(* IEC 61131-3 sources: repolevel_ST_code_completion/real_groud_truth最新/repoeval_plc_hello_mixing_tank/full_result, 6 files *)

(* ---- F_ResetDeviceCommands.st ---- *)
FUNCTION F_ResetDeviceCommands : BOOL
VAR_IN_OUT
	// HMI命令标志（需要复位）
	bMixerRunCmd		:	BOOL;
	bMixerStopCmd		:	BOOL;
	bMedium1OpenCmd		:	BOOL;
	bMedium1CloseCmd	:	BOOL;
	bMedium2OpenCmd		:	BOOL;
	bMedium2CloseCmd	:	BOOL;
	bDrainOpenCmd		:	BOOL;
	bDrainCloseCmd		:	BOOL;
END_VAR
VAR_INPUT
	// 设备状态反馈
	bMixerRunning		:	BOOL;
	bMedium1Opened		:	BOOL;
	bMedium2Opened		:	BOOL;
	bDrainOpened		:	BOOL;
END_VAR

VAR_OUTPUT
	// 复位完成标志
	bResetComplete		:	BOOL;
END_VAR

// 功能描述：复位所有HMI命令标志，当设备状态与命令一致时完成复位
bResetComplete := FALSE;

// 混合电机命令复位逻辑
IF NOT bMixerRunning AND bMixerRunCmd THEN
	bMixerRunCmd := FALSE;
END_IF;

IF bMixerRunning AND bMixerStopCmd THEN
	bMixerStopCmd := FALSE;
END_IF;

// Medium1命令复位逻辑
IF NOT bMedium1Opened AND bMedium1OpenCmd THEN
	bMedium1OpenCmd := FALSE;
END_IF;

IF bMedium1Opened AND bMedium1CloseCmd THEN
	bMedium1CloseCmd := FALSE;
END_IF;

// Medium2命令复位逻辑
IF NOT bMedium2Opened AND bMedium2OpenCmd THEN
	bMedium2OpenCmd := FALSE;
END_IF;

IF bMedium2Opened AND bMedium2CloseCmd THEN
	bMedium2CloseCmd := FALSE;
END_IF;

// Drain命令复位逻辑
IF NOT bDrainOpened AND bDrainOpenCmd THEN
	bDrainOpenCmd := FALSE;
END_IF;

IF bDrainOpened AND bDrainCloseCmd THEN
	bDrainCloseCmd := FALSE;
END_IF;

// 检查是否所有命令标志已复位
IF NOT bMixerRunCmd AND NOT bMixerStopCmd AND
   NOT bMedium1OpenCmd AND NOT bMedium1CloseCmd AND
   NOT bMedium2OpenCmd AND NOT bMedium2CloseCmd AND
   NOT bDrainOpenCmd AND NOT bDrainCloseCmd THEN
	bResetComplete := TRUE;
END_IF;

RETURN bResetComplete;
END_FUNCTION

(* ---- F_UpdateLimitSwitches.st ---- *)
FUNCTION F_UpdateLimitSwitches : BOOL
VAR_INPUT
	rTankLevel			:	REAL;			// 当前液位 (%)
	rFullThreshold		:	REAL := 85.0;	// 满液位阈值 (%)
	rEmptyThreshold		:	REAL := 5.0;	// 空液位阈值 (%)
END_VAR
VAR_OUTPUT
	bLevelFull			:	BOOL;			// 液位满开关
	bLevelEmpty			:	BOOL;			// 液位空开关
END_VAR

# --------------------------------------------------
# FUNCTION F_UpdateLimitSwitches
# This function updates the limit switches based on the current tank level.
# If the tank level exceeds the full threshold, the full switch is activated.
# If the tank level drops below the empty threshold, the empty switch is activated.
# --------------------------------------------------

# Update the full level switch
IF rTankLevel >= rFullThreshold THEN
    bLevelFull := TRUE;
ELSE
    bLevelFull := FALSE;
END_IF;

# Update the empty level switch
IF rTankLevel <= rEmptyThreshold THEN
    bLevelEmpty := TRUE;
ELSE
    bLevelEmpty := FALSE;
END_IF;

# Return TRUE to indicate the function executed successfully
F_UpdateLimitSwitches := TRUE;
END_FUNCTION

(* ---- FB_AutoSequence.st ---- *)
FUNCTION_BLOCK FB_AutoSequence
VAR_INPUT
	bEnable				:	BOOL;			// 使能自动序列
	bReset				:	BOOL;			// 复位到排空状态

	// 液位传感器反馈
	bTankLevelFull		:	BOOL;			// 液位满传感器
	bTankLevelEmpty		:	BOOL;			// 液位空传感器

	// 设备状态反馈
	bMixerRunning		:	BOOL;			// 混合电机运行中
	bMedium1Opened		:	BOOL;			// 介质1阀门打开
	bMedium2Opened		:	BOOL;			// 介质2阀门打开
	bDrainOpened		:	BOOL;			// 排空阀门打开

	// 配置参数
	tMixingDuration		:	TIME := T#10S;	// 混合持续时间
END_VAR
VAR_OUTPUT
	// 设备控制输出
	bMixerRunCmd		:	BOOL;			// 混合电机运行命令
	bMedium1OpenCmd		:	BOOL;			// 介质1阀门打开命令
	bMedium2OpenCmd		:	BOOL;			// 介质2阀门打开命令
	bDrainOpenCmd		:	BOOL;			// 排空阀门打开命令

	// 状态输出
	eCurrentState		:	AUTO_SEQUENCE;	// 当前状态
	nCyclesCompleted	:	UINT;			// 完成的循环次数
END_VAR

VAR
	// 内部状态变量
	eNextState			:	AUTO_SEQUENCE;	// 下一个状态
	tStateTimer			:	TIME;			// 状态计时器
	nCycleCounter		:	UINT := 0;		// 循环计数器
	bTransitionFlag		:	BOOL := FALSE;	// 状态转换标志
END_VAR

// 自动序列状态枚举
TYPE AUTO_SEQUENCE :
(
	IDLE,				// 空闲状态
	FILLING_MEDIUM1,	// 介质1填充状态
	FILLING_MEDIUM2,	// 介质2填充状态
	MIXING,				// 混合状态
	DRAINING			// 排空状态
);
END_TYPE

// 自动序列逻辑实现
IF bEnable THEN
	CASE eCurrentState OF
		IDLE:
			IF bTankLevelEmpty THEN
				eNextState := FILLING_MEDIUM1;
			END_IF;

		FILLING_MEDIUM1:
			bMedium1OpenCmd := TRUE;
			IF bTankLevelFull THEN
				bMedium1OpenCmd := FALSE;
				eNextState := FILLING_MEDIUM2;
			END_IF;

		FILLING_MEDIUM2:
			bMedium2OpenCmd := TRUE;
			IF bTankLevelFull THEN
				bMedium2OpenCmd := FALSE;
				eNextState := MIXING;
			END_IF;

		MIXING:
			bMixerRunCmd := TRUE;
			IF tStateTimer >= tMixingDuration THEN
				bMixerRunCmd := FALSE;
				eNextState := DRAINING;
			END_IF;

		DRAINING:
			bDrainOpenCmd := TRUE;
			IF bTankLevelEmpty THEN
				bDrainOpenCmd := FALSE;
				eNextState := IDLE;
				nCycleCounter := nCycleCounter + 1;
			END_IF;
	END_CASE;

	// 状态更新
	IF eNextState <> eCurrentState THEN
		eCurrentState := eNextState;
		tStateTimer := T#0S; // 重置状态计时器
	END_IF;

	// 状态计时器更新
	tStateTimer := tStateTimer + T#1MS;
ELSE
	// 禁用时复位所有命令和状态
	bMixerRunCmd := FALSE;
	bMedium1OpenCmd := FALSE;
	bMedium2OpenCmd := FALSE;
	bDrainOpenCmd := FALSE;
	eCurrentState := IDLE;
	nCycleCounter := 0;
END_IF;

IF bReset THEN
	// 复位逻辑
	bMixerRunCmd := FALSE;
	bMedium1OpenCmd := FALSE;
	bMedium2OpenCmd := FALSE;
	bDrainOpenCmd := FALSE;
	eCurrentState := IDLE;
	nCycleCounter := 0;
	tStateTimer := T#0S;
END_IF;
END_FUNCTION_BLOCK

(* ---- FB_ManualControl.st ---- *)
FUNCTION_BLOCK FB_ManualControl
VAR_INPUT
	// HMI命令输入
	bMixerRunCmd		:	BOOL;
	bMixerStopCmd		:	BOOL;
	bMedium1OpenCmd		:	BOOL;
	bMedium1CloseCmd	:	BOOL;
	bMedium2OpenCmd		:	BOOL;
	bMedium2CloseCmd	:	BOOL;
	bDrainOpenCmd		:	BOOL;
	bDrainCloseCmd		:	BOOL;

	// 设备反馈输入
	bMixerRunning		:	BOOL;
	bMedium1Opened		:	BOOL;
	bMedium2Opened		:	BOOL;
	bDrainOpened		:	BOOL;
END_VAR
VAR_OUTPUT
	// 设备控制输出
	bMixerRunCmdOut		:	BOOL;
	bMedium1OpenCmdOut	:	BOOL;
	bMedium2OpenCmdOut	:	BOOL;
	bDrainOpenCmdOut	:	BOOL;
END_VAR

VAR
	// 内部变量
	bResetCommands		:	BOOL;
END_VAR

// 主程序逻辑
// 复位命令逻辑
bResetCommands := F_ResetDeviceCommands(
	bMixerRunCmd := bMixerRunCmd,
	bMixerStopCmd := bMixerStopCmd,
	bMedium1OpenCmd := bMedium1OpenCmd,
	bMedium1CloseCmd := bMedium1CloseCmd,
	bMedium2OpenCmd := bMedium2OpenCmd,
	bMedium2CloseCmd := bMedium2CloseCmd,
	bDrainOpenCmd := bDrainOpenCmd,
	bDrainCloseCmd := bDrainCloseCmd,
	bMixerRunning := bMixerRunning,
	bMedium1Opened := bMedium1Opened,
	bMedium2Opened := bMedium2Opened,
	bDrainOpened := bDrainOpened
);

// 输出命令逻辑
IF bMixerRunCmd AND NOT bMixerRunning THEN
	bMixerRunCmdOut := TRUE;	// 启动混合电机
ELSE
	bMixerRunCmdOut := FALSE;
END_IF

IF bMedium1OpenCmd AND NOT bMedium1Opened THEN
	bMedium1OpenCmdOut := TRUE;	// 打开介质1阀门
ELSE
	bMedium1OpenCmdOut := FALSE;
END_IF

IF bMedium2OpenCmd AND NOT bMedium2Opened THEN
	bMedium2OpenCmdOut := TRUE;	// 打开介质2阀门
ELSE
	bMedium2OpenCmdOut := FALSE;
END_IF

IF bDrainOpenCmd AND NOT bDrainOpened THEN
	bDrainOpenCmdOut := TRUE;	// 打开排空阀门
ELSE
	bDrainOpenCmdOut := FALSE;
END_IF
END_FUNCTION_BLOCK

(* ---- FB_ModeController.st ---- *)
FUNCTION_BLOCK FB_ModeController
VAR_INPUT
	bSetToAuto		:	BOOL;	// 切换到自动模式命令
	bSetToManual	:	BOOL;	// 切换到手动模式命令
END_VAR
VAR_OUTPUT
	eCurrentMode	:	MODES;	// 当前模式
	bModeChanged	:	BOOL;	// 模式改变标志
END_VAR

VAR
	ePreviousMode	:	MODES;	// 上一次模式
END_VAR

// 定义模式类型
TYPE MODES : (MANUAL, AUTO);
END_TYPE

// 初始化
IF NOT eCurrentMode THEN
	eCurrentMode := MANUAL; // 默认模式为手动模式
	ePreviousMode := MANUAL;
	bModeChanged := FALSE;
END_IF

// 模式切换逻辑
IF bSetToAuto AND (eCurrentMode <> AUTO) THEN
	ePreviousMode := eCurrentMode;
	eCurrentMode := AUTO;
	bModeChanged := TRUE;
ELSIF bSetToManual AND (eCurrentMode <> MANUAL) THEN
	ePreviousMode := eCurrentMode;
	eCurrentMode := MANUAL;
	bModeChanged := TRUE;
ELSE
	bModeChanged := FALSE;
END_IF
END_FUNCTION_BLOCK

(* ---- FB_TankLevelSimulator.st ---- *)
FUNCTION_BLOCK FB_TankLevelSimulator
VAR_INPUT
	bMedium1Opened		:	BOOL;			// 介质1阀门打开
	bMedium2Opened		:	BOOL;			// 介质2阀门打开
	bDrainOpened		:	BOOL;			// 排空阀门打开
	bReset				:	BOOL;			// 复位到初始液位

	// 配置参数
	rInitialLevel		:	REAL := 25.0;	// 初始液位 (%)
	rFillRate1			:	REAL := 0.1;	// 介质1填充速率 (%/cycle)
	rFillRate2			:	REAL := 0.1;	// 介质2填充速率 (%/cycle)
	rDrainRate			:	REAL := 0.2;	// 排空速率 (%/cycle)
	rMinLevel			:	REAL := 0.0;	// 最小液位 (%)
	rMaxLevel			:	REAL := 100.0;	// 最大液位 (%)
END_VAR
VAR_OUTPUT
	rCurrentLevel		:	REAL;			// 当前液位 (%)
END_VAR

VAR
	rLevel				:	REAL;			// 内部液位变量
END_VAR

// 初始化液位
IF bReset THEN
	rLevel := rInitialLevel;
END_IF

// 液位计算逻辑
IF bMedium1Opened THEN
	rLevel := rLevel + rFillRate1;
END_IF

IF bMedium2Opened THEN
	rLevel := rLevel + rFillRate2;
END_IF

IF bDrainOpened THEN
	rLevel := rLevel - rDrainRate;
END_IF

// 限制液位范围
IF rLevel < rMinLevel THEN
	rLevel := rMinLevel;
ELSIF rLevel > rMaxLevel THEN
	rLevel := rMaxLevel;
END_IF

// 输出当前液位
rCurrentLevel := rLevel;
END_FUNCTION_BLOCK
